PROGRAM FBD_Assign_IO
VAR
	fbButtonBox: FB_ButtonBox;
	fbMotorControl: FB_MotorControl;
END_VAR

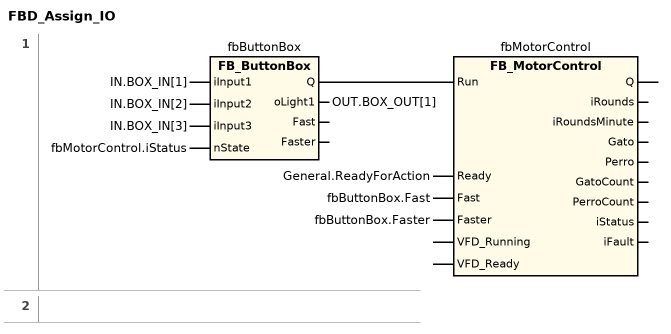
// NETWORK 1
fbButtonBox(
    iInput1 := IN.BOX_IN[1],
    iInput2 := IN.BOX_IN[2],
    iInput3 := IN.BOX_IN[3],
    nState := fbMotorControl.iStatus,
    oLight1 => OUT.BOX_OUT[1]); // FB_ButtonBox
fbMotorControl(
    Run := fbButtonBox.Q,
    Ready := General.ReadyForAction,
    Fast := fbButtonBox.Fast,
    Faster := fbButtonBox.Faster); // FB_MotorControl

// NETWORK 2

END_PROGRAM

(* stored: Version 1.1.0.1, ProductVersion 3.1.4024.10
   POU FBD_Assign_IO: Id {5015793d-548e-4713-ad62-be76714ca000}, SpecialFunc None *)
